Staubli VAL3: rollsum.pgx

public program rollsum(num& x_nInput[], num x_nWindow, num& x_nResult[])
  local num l_nLength
  local num l_nElement
  local num l_nSum
begin

  l_nLength = size(x_nInput)
  x_nResult = 0
  resize(x_nResult,1,l_nLength-x_nWindow+1)

  l_nElement = 0
  while l_nElement <l_nLength-x_nWindow+1
    call utils:range(l_nElement, l_nElement+x_nWindow, 1,nIndex)
    call utils:extractNum(x_nInput,nIndex,nResult)
    call sum(nResult, l_nSum)

    x_nResult[l_nElement] = l_nSum
    l_nElement = l_nElement + 1
  endWhile

end
